// TwinCAT 3 PLC project Untitled1
// ProgramVersion: 3.1.4023.0
// libraries:
//   Tc2_Standard, * (Beckhoff Automation GmbH)
//   Tc2_System, * (Beckhoff Automation GmbH)
//   Tc3_Module, * (Beckhoff Automation GmbH)
// project tree:
//   GVLs/ Grinder.TcGVL
//   / PlcTask.TcTTO
//   POUs/ MAIN.TcPOU, RunGrindingWheel.TcPOU
// real-time tasks:
//   TASK PlcTask: cycle T#10ms, priority 20, ADS port 350

CONFIGURATION Untitled1
    RESOURCE PLC ON TwinCAT3
        TASK PlcTask(INTERVAL := T#10ms, PRIORITY := 20);
        PROGRAM MAIN WITH PlcTask : MAIN;
    END_RESOURCE
END_CONFIGURATION

// ---- GVLs/Grinder.TcGVL
{attribute 'qualified_only'}
VAR_GLOBAL
	GrindingWheelMS AT %Q* : BOOL;
	StartGrindingWheelPB AT %I* : BOOL;
	StopGrindingWheelPB AT %I*  : BOOL;	
END_VAR

// ---- POUs/MAIN.TcPOU
PROGRAM MAIN
VAR
END_VAR

RunGrindingWheel ();

END_PROGRAM

// ---- POUs/RunGrindingWheel.TcPOU
PROGRAM RunGrindingWheel
VAR
END_VAR

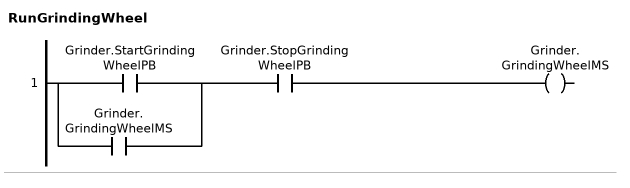
// NETWORK 1
Grinder.GrindingWheelMS := (Grinder.StartGrindingWheelPB OR Grinder.GrindingWheelMS) AND Grinder.StopGrindingWheelPB;

END_PROGRAM
